(* Schneider Machine Expert - Basic project first in priority system, file version 2.7.0.0 *)
(* ProjectInformations: Name=New project *)

HARDWARE
  Cpu 0: TM221M16R/G
  EthernetConfiguration: NetworkName=M221, IpAllocationMode=FixedAddress, IpAddress=0.0.0.0, SubnetMask=0.0.0.0
  SerialLineConfiguration: Baud=Baud19200, Parity=ParityEven, DataBits=DataBits8, StopBits=StopBits1, PhysicalMedium=PhysicalMediumRs485, TransmissionMode=TransmissionModeModbusRtu, SlaveId=1, Addressing=SlaveAddressing
  MastTask: UsePeriodScanMode=false, PeriodScan=100
  FastTask: Period=255
  CpuBehavior: StartingMode=StartAsPreviousState, AutoSaveRamOnEeprom=true, WatchdogPeriod=250

SYMBOLS  (address, symbol, comment, settings)
  %I0.0     PG1
  %I0.1     PG2
  %I0.2     HS1
  %I0.3     PF1
  %I0.4     PF2
  %I0.5     HOST
  %Q0.0     RESET
  %Q0.1     PG_LAMP
  %Q0.2     HS_LAMP
  %Q0.3     PF_LAMP

POU New POU
  (* SectionNumber=0 *)

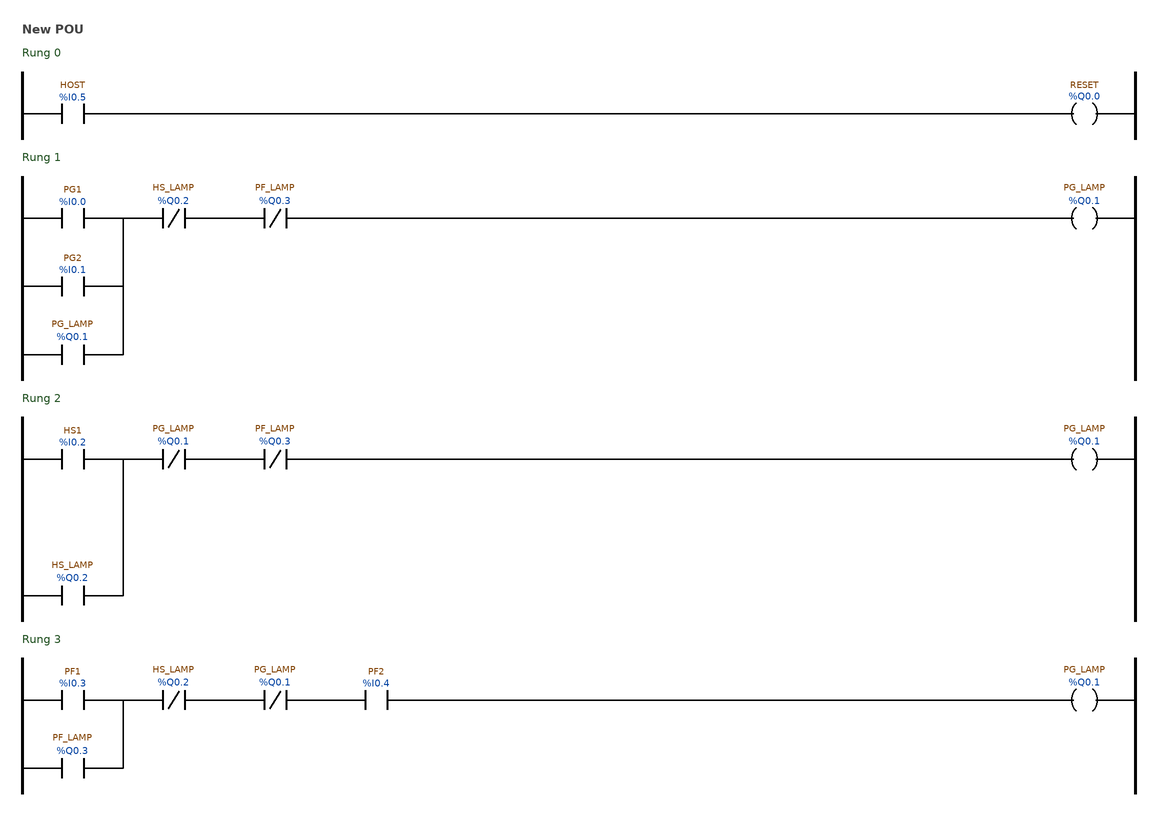

// Rung 0
  LD %I0.5                (* HOST *)
  ST %Q0.0                (* RESET *)
  // as ST:
  //   RESET := HOST;

// Rung 1
  LD %I0.0                (* PG1 *)
  OR %I0.1                (* PG2 *)
  OR %Q0.1                (* PG_LAMP *)
  ANDN %Q0.2              (* HS_LAMP *)
  ANDN %Q0.3              (* PF_LAMP *)
  ST %Q0.1                (* PG_LAMP *)
  // as ST:
  //   PG_LAMP := (PG1 OR PG2 OR PG_LAMP) AND NOT HS_LAMP AND NOT PF_LAMP;

// Rung 2
  LD %I0.2                (* HS1 *)
  OR %Q0.2                (* HS_LAMP *)
  ANDN %Q0.1              (* PG_LAMP *)
  ANDN %Q0.3              (* PF_LAMP *)
  ST %Q0.1                (* PG_LAMP *)
  // as ST:
  //   PG_LAMP := (HS1 OR HS_LAMP) AND NOT PG_LAMP AND NOT PF_LAMP;

// Rung 3
  LD %I0.3                (* PF1 *)
  OR %Q0.3                (* PF_LAMP *)
  ANDN %Q0.2              (* HS_LAMP *)
  ANDN %Q0.1              (* PG_LAMP *)
  AND %I0.4               (* PF2 *)
  ST %Q0.1                (* PG_LAMP *)
  // as ST:
  //   PG_LAMP := (PF1 OR PF_LAMP) AND NOT HS_LAMP AND NOT PG_LAMP AND PF2;
